Fanuc KAREL source: kf00080.KL

PROGRAM KF00080
%STACKSIZE=65535
%PRIORITY=65535
%NOLOCKGROUP
VAR
I : INTEGER
J : INTEGER
X : REAL
Y : REAL
B : BOOLEAN
C : BOOLEAN
TXT : STRING[80]
TXT2 : STRING[80]
AI : ARRAY[4] OF INTEGER
BI : ARRAY[4] OF INTEGER
P : XYZWPR
JP : JOINTPOS9
PF : POSITION
V1 : VECTOR
V2 : VECTOR
STATUS : INTEGER
-- UNRESOLVED DECLARATIONS (source type spelling not recovered)
-- QT : TYPE_0x1100 (type_u16=0x1100)
BEGIN
INIT_QUEUE(QT)
END KF00080
